FUNCTION F_CommandAllSequences : BOOL
VAR_IN_OUT
	itfSequenceArray	: ARRAY[*] OF ITF_ModuleSequenceControl;
END_VAR
VAR_INPUT
	eCommand			: E_ModuleSequenceCommand;
	nSubCount			: UDINT;
END_VAR
VAR
	i:	UDINT;
END_VAR

CASE eCommand OF
	E_ModuleSequenceCommand.Begin:
		FOR i := 1 TO nSubCount DO
			itfSequenceArray[i].BeginSequence();
		END_FOR
		
	E_ModuleSequenceCommand.Block:
		FOR i := 1 TO nSubCount DO
			itfSequenceArray[i].BlockSequence();
		END_FOR
	
	E_ModuleSequenceCommand.Resume:
		FOR i := 1 TO nSubCount DO
			itfSequenceArray[i].ResumeSequence();
		END_FOR
	
	E_ModuleSequenceCommand.Revert:
		FOR i := 1 TO nSubCount DO
			itfSequenceArray[i].RevertSequence();
		END_FOR
	
	E_ModuleSequenceCommand.Cancel:
		FOR i := 1 TO nSubCount DO
			itfSequenceArray[i].CancelSequence();
		END_FOR
	
	E_ModuleSequenceCommand.Reiterate:
		FOR i := 1 TO nSubCount DO
			itfSequenceArray[i].ReiterateSequence();
		END_FOR
	
END_CASE

END_FUNCTION

(* stored: Version 1.1.0.1, ProductVersion 3.1.4024.9
   POU F_CommandAllSequences: Id {2a8ddc45-54b4-4d4f-af91-e4616bd76094}, SpecialFunc None *)
